// TIA Portal project "washingmachine" (V16)

(* hardware
DEVICE "S71500/ET200MP station_1"  S7-1500 station
   slot 0: "Rail_0"  Rack  6ES7 590-1***0-0AA0
   slot 1: "PLC_1"  CPU 1511C-1 PN  6ES7 511-1CK00-0AB0  V2.8
      slot 3: "CPU display_1"  6ES7591-1AA00-0AA0
      slot 32768: "PROFINET interface_1"  X1
         slot 32769: "Port_1"  X1 P1
         slot 32770: "Port_2"  X1 P2
      slot 34817: "Virtual CP interface port_1"  Virtual CP interface port  Virtual CP interface port
DEVICE "HMI_1"  TP900 Comfort
   slot 0: "HMI_1"  TP900 Comfort  6AV2 124-0JC01-0AX0  16.0.0.0
   slot 1: "HMI_RT_1"  TP900 Comfort  6AV2 124-0JC01-0AX0  16.0.0.0
   slot 5: "HMI_1.IE_CP_1"  PROFINET Interface  16.0.0.0
      slot 1: "PROFINET Interface_1"  PROFINET Interface
         slot 1: "Port_1"  Port
         slot 2: "Port_2"  Port
   slot 7: "HMI_1.MPI/DP_CP_1"  MPI/DP Interface  16.0.0.0
*)

// ===== PLC "PLC_1"  CPU 1511C-1 PN =====

VAR_GLOBAL   // PLC tag table "Default tag table"
   "Door is closed" AT %M0.0 : Bool;
   "Water Level MAx" AT %M0.1 : Bool;
   "Temperature Min" AT %M0.2 : Bool;
   "Water Level Min" AT %M0.3 : Bool;
   "Temperature Max" AT %M0.4 : Bool;
   "Start" AT %M0.5 : Bool;
   "Water İnlet" AT %M1.0 : Bool;
   "Heating" AT %M1.1 : Bool;
   "Water Outlet valve" AT %M1.2 : Bool;
   "Motor Switch" AT %M1.3 : Bool;
   "High Revolution" AT %M1.4 : Bool;
   "Change Direction" AT %M1.5 : Bool;
   "Door Lock" AT %M1.6 : Bool;
   "PTRIG3" AT %M2.0 : Bool;
   "start_basildi" AT %M3.0 : Bool;
   "NTRIG" AT %M2.1 : Bool;
   "PTRIG4" AT %M2.2 : Bool;
   "PTRIG5" AT %M2.3 : Bool;
   "PTRIG6" AT %M2.4 : Bool;
   "ROTA" AT %M2.5 : Bool;
   "PTRIG7" AT %M2.6 : Bool;
   "PTRIG8" AT %M2.7 : Bool;
   "Heating bitti" AT %M4.0 : Bool;
   "PTRIG 9" AT %M4.2 : Bool;
   "Sol" AT %M1.7 : Bool;
   "PTRIG10" AT %M4.3 : Bool;
   "Rota-Sol" AT %M4.4 : Bool;
   "Rota-sağ" AT %M4.5 : Bool;
   "PTRIG11" AT %M4.6 : Bool;
   "PTRIG12" AT %M4.7 : Bool;
   "PTRIG13" AT %M5.0 : Bool;
   "NTRIG2" AT %M5.2 : Bool;
   "dönüş bitti" AT %M5.4 : Bool;
   "PTRIG14" AT %M5.5 : Bool;
   "PTRIG15" AT %M5.6 : Bool;
   "PTRIG16" AT %M5.7 : Bool;
   "PTRIG17" AT %M6.0 : Bool;
   "Count" AT %M0.6 : Bool;
   "output" AT %M7.0 : Bool;
   "p_trig1" AT %M7.1 : Bool;
   "p_trig2" AT %M7.3 : Bool;
   "enable" AT %M0.7 : Bool;
   "enable2" AT %M3.1 : Bool;
END_VAR

// folder: System blocks/Program resources

DATA_BLOCK "IEC_Timer_0_DB"   // DB1
{ S7_Optimized_Access := 'TRUE' }
AUTHOR : Simatic
FAMILY : IEC
NAME : IEC_TMR
VERSION : 1.0
// stored: InstanceOfName IEC_TIMER
"IEC_TIMER"
BEGIN
END_DATA_BLOCK

DATA_BLOCK "IEC_Timer_0_DB1"   // DB2
{ S7_Optimized_Access := 'TRUE' }
AUTHOR : Simatic
FAMILY : IEC
NAME : IEC_TMR
VERSION : 1.0
// stored: InstanceOfName IEC_TIMER
"IEC_TIMER"
BEGIN
END_DATA_BLOCK

DATA_BLOCK "saga_donus_sayim"   // DB3
{ S7_Optimized_Access := 'TRUE' }
AUTHOR : Simatic
FAMILY : IEC
NAME : CNTR
VERSION : 1.0
// stored: InstanceOfName IEC_COUNTER
"IEC_COUNTER"
BEGIN
END_DATA_BLOCK

DATA_BLOCK "sola_donus_sayim"   // DB4
{ S7_Optimized_Access := 'TRUE' }
AUTHOR : Simatic
FAMILY : IEC
NAME : CNTR
VERSION : 1.0
// stored: InstanceOfName IEC_COUNTER
"IEC_COUNTER"
BEGIN
END_DATA_BLOCK

DATA_BLOCK "IEC_Timer_0_DB_1"   // DB5
{ S7_Optimized_Access := 'TRUE' }
AUTHOR : Simatic
FAMILY : IEC
NAME : IEC_TMR
VERSION : 1.0
// stored: InstanceOfName IEC_TIMER
"IEC_TIMER"
BEGIN
END_DATA_BLOCK

DATA_BLOCK "IEC_Timer_0_DB_2"   // DB6
{ S7_Optimized_Access := 'TRUE' }
AUTHOR : Simatic
FAMILY : IEC
NAME : IEC_TMR
VERSION : 1.0
// stored: InstanceOfName IEC_TIMER
"IEC_TIMER"
BEGIN
END_DATA_BLOCK

DATA_BLOCK "IEC_Counter_0_DB"   // DB7
{ S7_Optimized_Access := 'TRUE' }
AUTHOR : Simatic
FAMILY : IEC
NAME : CNTR
VERSION : 1.0
// stored: InstanceOfName IEC_COUNTER
"IEC_COUNTER"
BEGIN
END_DATA_BLOCK

DATA_BLOCK "IEC_Timer_0_DB_3"   // DB8
{ S7_Optimized_Access := 'TRUE' }
AUTHOR : Simatic
FAMILY : IEC
NAME : IEC_TMR
VERSION : 1.0
// stored: InstanceOfName IEC_TIMER
"IEC_TIMER"
BEGIN
END_DATA_BLOCK

// folder: (top level)

ORGANIZATION_BLOCK "Main"   // OB1, LAD, ProgramCycle
TITLE = "Main Program Sweep (Cycle)"
{ S7_Optimized_Access := 'TRUE' }
VERSION : 0.1
   VAR_INPUT
      Initial_Call : Bool;   // Initial call of this OB
      Remanence : Bool;   // =True, if remanent data are available
   END_VAR
   VAR_TEMP   // added for the SCL form of the ladder/FBD networks
      _w1 : Bool;
      _w2 : Bool;
      _w3 : Bool;
      _w4 : Bool;
   END_VAR
BEGIN

REGION Network 1
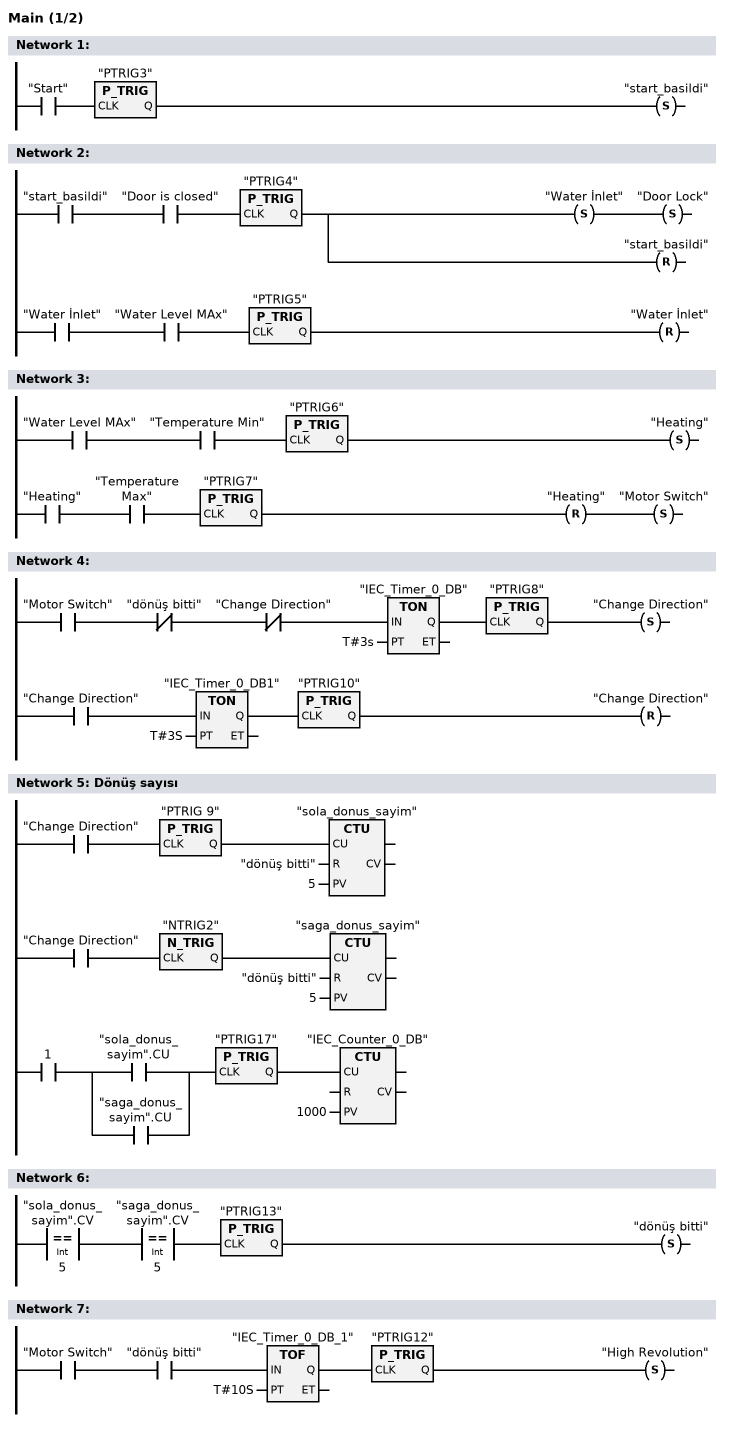
   RUNG wire#powerrail
      Contact( "Start" )
      P_Trig( "PTRIG3" )
      S_Coil( "start_basildi" )
   END_RUNG
   // the same network as SCL:
   #_w1 := "Start" AND NOT "PTRIG3";   // rising edge
   "PTRIG3" := "Start";
   IF #_w1 THEN "start_basildi" := TRUE; END_IF;
END_REGION

REGION Network 2
   RUNG wire#powerrail
      Contact( "start_basildi" )
      Contact( "Door is closed" )
      P_Trig( "PTRIG4" )
      wire#w1
      S_Coil( "Water İnlet" )
      S_Coil( "Door Lock" )
   END_RUNG
   RUNG wire#w1
      R_Coil( "start_basildi" )
   END_RUNG
   RUNG wire#powerrail
      Contact( "Water İnlet" )
      Contact( "Water Level MAx" )
      P_Trig( "PTRIG5" )
      R_Coil( "Water İnlet" )
   END_RUNG
   // the same network as SCL:
   #_w1 := "start_basildi" AND "Door is closed";
   #_w2 := #_w1 AND NOT "PTRIG4";   // rising edge
   "PTRIG4" := #_w1;
   IF #_w2 THEN
       "Water İnlet" := TRUE;
       "Door Lock" := TRUE;
       "start_basildi" := FALSE;
   END_IF;
   #_w3 := "Water İnlet" AND "Water Level MAx";
   #_w4 := #_w3 AND NOT "PTRIG5";   // rising edge
   "PTRIG5" := #_w3;
   IF #_w4 THEN "Water İnlet" := FALSE; END_IF;
END_REGION

REGION Network 3
   RUNG wire#powerrail
      Contact( "Water Level MAx" )
      Contact( "Temperature Min" )
      P_Trig( "PTRIG6" )
      S_Coil( "Heating" )
   END_RUNG
   RUNG wire#powerrail
      Contact( "Heating" )
      Contact( "Temperature Max" )
      P_Trig( "PTRIG7" )
      R_Coil( "Heating" )
      S_Coil( "Motor Switch" )
   END_RUNG
   // the same network as SCL:
   #_w1 := "Water Level MAx" AND "Temperature Min";
   #_w2 := #_w1 AND NOT "PTRIG6";   // rising edge
   "PTRIG6" := #_w1;
   IF #_w2 THEN "Heating" := TRUE; END_IF;
   #_w3 := "Heating" AND "Temperature Max";
   #_w4 := #_w3 AND NOT "PTRIG7";   // rising edge
   "PTRIG7" := #_w3;
   IF #_w4 THEN
       "Heating" := FALSE;
       "Motor Switch" := TRUE;
   END_IF;
END_REGION

REGION Network 4
   "IEC_Timer_0_DB".TON(IN := "Motor Switch" AND NOT "dönüş bitti" AND NOT "Change Direction", PT := T#3s);
   #_w1 := "IEC_Timer_0_DB".Q AND NOT "PTRIG8";   // rising edge
   "PTRIG8" := "IEC_Timer_0_DB".Q;
   IF #_w1 THEN "Change Direction" := TRUE; END_IF;
   "IEC_Timer_0_DB1".TON(IN := "Change Direction", PT := T#3S);
   #_w2 := "IEC_Timer_0_DB1".Q AND NOT "PTRIG10";   // rising edge
   "PTRIG10" := "IEC_Timer_0_DB1".Q;
   IF #_w2 THEN "Change Direction" := FALSE; END_IF;
END_REGION

REGION Network 5: Dönüş sayısı
   #_w1 := "Change Direction" AND NOT "PTRIG 9";   // rising edge
   "PTRIG 9" := "Change Direction";
   "sola_donus_sayim".CTU(CU := #_w1, R := "dönüş bitti", PV := 5);
   #_w2 := NOT "Change Direction" AND "NTRIG2";   // falling edge
   "NTRIG2" := "Change Direction";
   "saga_donus_sayim".CTU(CU := #_w2, R := "dönüş bitti", PV := 5);
   #_w3 := 1 AND ("sola_donus_sayim".CU OR "saga_donus_sayim".CU);
   #_w4 := #_w3 AND NOT "PTRIG17";   // rising edge
   "PTRIG17" := #_w3;
   "IEC_Counter_0_DB".CTU(CU := #_w4, PV := 1000);
END_REGION

REGION Network 6
   RUNG wire#powerrail
      { S7_Templates := "SrcType := Int" } EQ_Contact(in1 := "sola_donus_sayim".CV, in2 := 5)
      { S7_Templates := "SrcType := Int" } EQ_Contact(in1 := "saga_donus_sayim".CV, in2 := 5)
      P_Trig( "PTRIG13" )
      S_Coil( "dönüş bitti" )
   END_RUNG
   // the same network as SCL:
   #_w1 := ("sola_donus_sayim".CV = 5) AND ("saga_donus_sayim".CV = 5);
   #_w2 := #_w1 AND NOT "PTRIG13";   // rising edge
   "PTRIG13" := #_w1;
   IF #_w2 THEN "dönüş bitti" := TRUE; END_IF;
END_REGION

REGION Network 7
   "IEC_Timer_0_DB_1".TOF(IN := "Motor Switch" AND "dönüş bitti", PT := T#10S);
   #_w1 := "IEC_Timer_0_DB_1".Q AND NOT "PTRIG12";   // rising edge
   "PTRIG12" := "IEC_Timer_0_DB_1".Q;
   IF #_w1 THEN "High Revolution" := TRUE; END_IF;
END_REGION

REGION Network 8
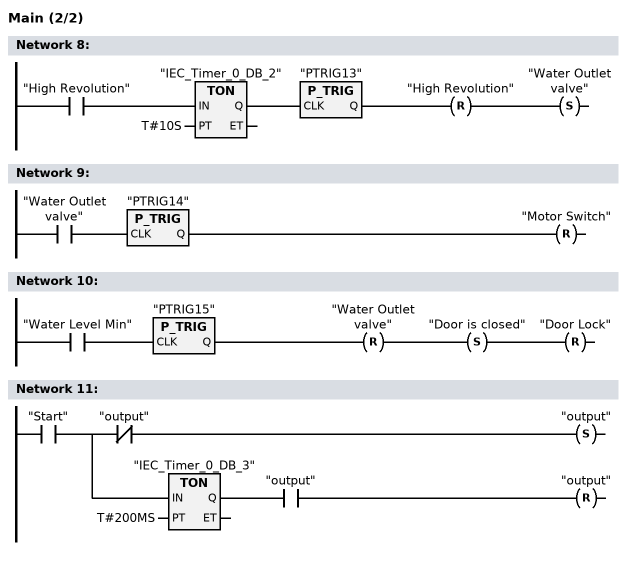
   "IEC_Timer_0_DB_2".TON(IN := "High Revolution", PT := T#10S);
   #_w1 := "IEC_Timer_0_DB_2".Q AND NOT "PTRIG13";   // rising edge
   "PTRIG13" := "IEC_Timer_0_DB_2".Q;
   IF #_w1 THEN
       "High Revolution" := FALSE;
       "Water Outlet valve" := TRUE;
   END_IF;
END_REGION

REGION Network 9
   RUNG wire#powerrail
      Contact( "Water Outlet valve" )
      P_Trig( "PTRIG14" )
      R_Coil( "Motor Switch" )
   END_RUNG
   // the same network as SCL:
   #_w1 := "Water Outlet valve" AND NOT "PTRIG14";   // rising edge
   "PTRIG14" := "Water Outlet valve";
   IF #_w1 THEN "Motor Switch" := FALSE; END_IF;
END_REGION

REGION Network 10
   RUNG wire#powerrail
      Contact( "Water Level Min" )
      P_Trig( "PTRIG15" )
      R_Coil( "Water Outlet valve" )
      S_Coil( "Door is closed" )
      R_Coil( "Door Lock" )
   END_RUNG
   // the same network as SCL:
   #_w1 := "Water Level Min" AND NOT "PTRIG15";   // rising edge
   "PTRIG15" := "Water Level Min";
   IF #_w1 THEN
       "Water Outlet valve" := FALSE;
       "Door is closed" := TRUE;
       "Door Lock" := FALSE;
   END_IF;
END_REGION

REGION Network 11
   IF "Start" AND NOT "output" THEN "output" := TRUE; END_IF;
   "IEC_Timer_0_DB_3".TON(IN := "Start", PT := T#200MS);
   IF "IEC_Timer_0_DB_3".Q AND "output" THEN "output" := FALSE; END_IF;
END_REGION
END_ORGANIZATION_BLOCK

(* ===== HMI "HMI_RT_1" =====
system functions are stored by id; their names below are inferred from use
connection "HMI_Connection_1": ETHERNET, S7_1500_OMS

HMI tags "Default tag table"
   "Door is closed" : Bool = PLC "Door is closed" AT %M0.0, 1 s
   "Water Level MAx" : Bool = PLC "Water Level MAx" AT %M0.1, 1 s
   "Water Level Min" : Bool = PLC "Water Level Min" AT %M0.3, 1 s
   "Temperature Max" : Bool = PLC "Temperature Max" AT %M0.4, 1 s
   "Temperature Min" : Bool = PLC "Temperature Min" AT %M0.2, 1 s
   "Change Direction" : Bool = PLC "Change Direction" AT %M1.5, 1 s
   "High Revolution" : Bool = PLC "High Revolution" AT %M1.4, 1 s
   "Water İnlet" : Bool = PLC "Water İnlet" AT %M1.0, 1 s
   "Heating" : Bool = PLC Heating AT %M1.1, 1 s
   "Water Outlet valve" : Bool = PLC "Water Outlet valve" AT %M1.2, 1 s
   "Motor Switch" : Bool = PLC "Motor Switch" AT %M1.3, 1 s
   "Door Lock" : Bool = PLC "Door Lock" AT %M1.6, 1 s
   "Start" : Bool = PLC Start AT %M0.5, 1 s
   "Count" : Bool = PLC Count AT %M0.6, 1 s
   "IEC_Counter_0_DB_QU" : Bool = PLC IEC_Counter_0_DB.QU, 1 s
   "IEC_Counter_0_DB_CV" : Int = PLC IEC_Counter_0_DB.CV, 1 s

screen "Root screen" 800x420, template "Template_1"
   on GenerateScreen: SetTag("Start", 1)
   TextField "Text field_1" at 77,29 size 14x20; Text 'Text'
   Button "Button_1" at 16,76 size 125x32; TextOff 'Door is Closed'
      on Press: InvertBit("Door is closed")
   Button "Button_2" at 16,127 size 129x32; TextOff 'Water Level Max.'
      on Press: InvertBit("Water Level MAx")
   Button "Button_3" at 16,179 size 129x32; TextOff 'Water Level Min.'
      on Press: InvertBit("Water Level Min")
   Button "Button_4" at 16,230 size 129x32; TextOff 'Temperature Max'
      on Press: InvertBit("Temperature Max")
   Button "Button_5" at 16,282 size 129x32; TextOff 'Temperature Min'
      on Press: InvertBit("Temperature Min")
   Button "Button_6" at 16,25 size 130x32; TextOff 'Start'
      on Press: function_b14e0dd5("Start", 0)
   Circle "Circle_1" at 171,25 size 37x37
      Appearance <- "Start"
   Circle "Circle_2" at 171,75 size 37x37
      Appearance <- "Door is closed"
   Circle "Circle_3" at 171,126 size 37x37
      Appearance <- "Water Level MAx"
   Circle "Circle_4" at 171,177 size 37x37
      Appearance <- "Water Level Min"
   Circle "Circle_5" at 171,228 size 37x37
      Appearance <- "Temperature Max"
   Circle "Circle_6" at 171,279 size 37x37
      Appearance <- "Temperature Min"
   TextField "Text field_2" at 487,29 size 102x20; Text 'Water Inlet :'
   Circle "Circle_7" at 655,28 size 37x37
      Appearance <- "Water İnlet"
   TextField "Text field_3" at 487,70 size 62x20; Text 'Heating'
   Circle "Circle_8" at 655,69 size 37x37
      Appearance <- "Heating"
   TextField "Text field_4" at 487,112 size 159x20; Text 'Water Outlet Valve :'
   Circle "Circle_9" at 655,110 size 37x37
      Appearance <- "Water Outlet valve"
   TextField "Text field_5" at 487,153 size 103x20; Text 'Motor Switch'
   Circle "Circle_11" at 655,152 size 37x37
      Appearance <- "Motor Switch"
   TextField "Text field_6" at 487,236 size 121x20; Text 'High Revolution'
   Circle "Circle_10" at 655,193 size 37x37
      Appearance <- "Door Lock"
   TextField "Text field_7" at 487,195 size 92x20; Text 'Door locked'
   TextField "Text field_8" at 487,278 size 131x20; Text 'Change Direction'
   Circle "Circle_12" at 655,234 size 37x37
      Appearance <- "High Revolution"
   Circle "Circle_13" at 655,276 size 37x37
      Appearance <- "Change Direction"
   TextField "Text field_9" at 256,312 size 64x20; Text 'Count :'
   IOField "I/O field_1" at 339,313 size 96x32; FormatPattern s99999
      ProcessValue <- "IEC_Counter_0_DB_CV"

Template "Template_1" 800x420
   Button "Exit" at 720,360 size 78x58; TextOff 'Exit'; PictureOff "ExitRuntime_TP900_Comfort_TR"; PictureOn "ExitRuntime_TP900_Comfort_TR"
      on Release: StopRuntime(0)
   Button "Template_Button" at 640,360 size 78x58; TextOff 'Text'
   Button "Template_Button_1" at 560,360 size 78x58; TextOff 'Text'
   Button "Template_Button_2" at 480,360 size 78x58; TextOff 'Text'
   Button "Template_Button_3" at 400,360 size 78x58; TextOff 'Text'
   Button "Template_Button_4" at 321,360 size 78x58; TextOff 'Text'
   Button "Template_Button_5" at 241,360 size 78x58; TextOff 'Text'
   Button "Template_Button_6" at 161,360 size 78x58; TextOff 'Text'
   Button "Alarms" at 81,360 size 78x58; TextOff 'Alarms'; PictureOff "AlarmDisplay_TP900_Comfort_TR"; PictureOn "AlarmDisplay_TP900_Comfort_TR"
      on Release: function_ef3f5d25("Alarm window_Unacknowledged", -1)
   Button "Start screen" at 1,360 size 78x58; TextOff 'Start screen'; PictureOff "NavigateHome_TP900_Comfort_TR"; PictureOn "NavigateHome_TP900_Comfort_TR"
      on Release: ActivateScreen("Root screen", 0)
*)